FUNCTION_BLOCK FB_A_HKSystem IMPLEMENTS I_HKSystem
VAR_INPUT
	I_bVerbunden	:BOOL;		// Angabe ob HK-System angeschlossen ist
	I_iModus		:INT;		// Zustand des Systems (z.B. 0 = AUS | 1 = MAN | 2 = AUTO)
	I_iTemp			:INT;		// Aktuelle Temperatur um Heizmodus auszuwählen und zu stoppen
	I_bVerriegeln	:BOOL;		// Verriegelte Elemente sind nicht ansteuerbar
	I_bReset		:BOOL;		// Zustand des Baustein wird zurückgesetzt 
END_VAR

VAR_OUTPUT
	O_bPumpen		:BOOL;		// Pumpe des HK-Systems wird betrieben
	O_bKuehlen		:BOOL;		// HK-System heizt das Medium auf
	O_bHeizen		:BOOL;		// HK-System kühlt das Medium ab
	O_bStoerung		:BOOL;		// Befindet sich das Element in einem Error
	O_iStoerungID	:INT;		// Anzeigen von Störung über eine INT-Variable
	
END_VAR
	
VAR
	V_DefTemp		:INT;		// Variable für internes handling der Eigenschaft 
	V_Zeit			:TIME;		// Variable für internes handling der Eigenschaft 
	V_Zustand		:INT;		// Variable für internes handling der Eigenschaft 
	
	V_Timer			:TON;		// Runtime des Bausteins ermitteln
END_VAR

// Setzen der internen Variablen
V_Zeit := P_Laufzeit;
V_Zustand := P_Zustand;

// Fehler durch Verbindungsabbruch
IF O_bPumpen OR O_bKuehlen OR O_bHeizen THEN
	IF NOT I_bVerbunden THEN
		O_bPumpen := FALSE;
		O_bKuehlen := FALSE;
		O_bHeizen := FALSE;
		
		O_bStoerung := TRUE;
		O_iStoerungID := 04;
	END_IF
END_IF

// Abbruch des Heiz-Kühlprozesses beim erreichen der Temp
IF O_bHeizen OR O_bKuehlen THEN 
	IF I_iTemp = V_DefTemp THEN
		O_bKuehlen := FALSE;
		O_bHeizen := FALSE;		
	END_IF
END_IF

// Reset des Bausteins
IF I_bReset THEN
	O_bStoerung := FALSE;
	O_iStoerungID := 0;
END_IF

METHOD M_A_HK_AN : BOOL
VAR_INPUT
END_VAR
// EBENE 1: Verriegelung
IF NOT I_bVerriegeln THEN	
	// EBENE 2: AUTO-Modus
		IF I_iModus = 2 THEN
			// EBENE 3: Ist Pumpe AN
				IF O_bPumpen THEN
				// EBENE 4: Heizen oder Kühlen
					IF V_DefTemp > I_iTemp THEN
						O_bKuehlen := FALSE;
						O_bHeizen := TRUE;
						
						M_A_HK_AN := O_bHeizen;
						
					ELSIF I_iTemp > V_DefTemp THEN 	
						O_bHeizen := FALSE;
						O_bKuehlen := TRUE;
						
						M_A_HK_AN := O_bKuehlen;
					END_IF
				ELSE // Error: System ist nicht eingeschalten
					O_bStoerung := 1;
					O_iStoerungID := 11; 
				END_IF
			END_IF
END_IF
END_METHOD

METHOD M_A_HK_AUS : BOOL
VAR_INPUT
END_VAR
// EBENE 1: Verriegelung
IF NOT I_bVerriegeln THEN
		O_bKuehlen := FALSE;
		O_bHeizen := FALSE;
END_IF

IF O_bKuehlen = FALSE THEN
	M_A_HK_AUS := TRUE;
END_IF
END_METHOD

METHOD M_A_PUMPE_AN : BOOL
VAR_INPUT
END_VAR
// EBENE 1: Verriegelung
IF NOT I_bVerriegeln THEN	
	// EBENE 2: AUTO-Modus
		IF I_iModus = 2 THEN
			// EBENE 3: System muss angeschlossen sein
			IF I_bVerbunden THEN
				O_bPumpen := TRUE;
			ELSE 	// Error: System ist nicht angeschlossen
				O_bStoerung := 1;
				O_iStoerungID := 03;
			END_IF
		END_IF
END_IF

M_A_PUMPE_AN := O_bPumpen;
END_METHOD

METHOD M_A_PUMPE_AUS : BOOL
VAR_INPUT
END_VAR
// EBENE 1: Verriegelung
IF NOT I_bVerriegeln THEN
	IF NOT O_bHeizen AND NOT O_bKuehlen THEN
		O_bPumpen := FALSE;
	ELSE
		O_bStoerung := TRUE;
		O_iStoerungID := 05;
	END_IF
END_IF

IF O_bPumpen = FALSE THEN
	M_A_PUMPE_AUS := TRUE;
END_IF
END_METHOD

METHOD M_M_HK_AN : BOOL
VAR_INPUT
END_VAR
// EBENE 1: Verriegelung
IF NOT I_bVerriegeln THEN	
	// EBENE 2: MAN-Modus
		IF I_iModus = 1 THEN
			// EBENE 3: Ist Pumpe AN
				IF O_bPumpen THEN
				// EBENE 4: Heizen oder Kühlen
					IF V_DefTemp > I_iTemp THEN
						O_bKuehlen := FALSE;
						O_bHeizen := TRUE;
						
						M_M_HK_AN := O_bHeizen;
						
					ELSIF I_iTemp > V_DefTemp THEN 	
						O_bHeizen := FALSE;
						O_bKuehlen := TRUE;
						
						M_M_HK_AN := O_bKuehlen;
					END_IF
				ELSE // Error: System ist nicht eingeschalten
				O_bStoerung := 1;
				O_iStoerungID := 11; 	
				END_IF
			END_IF
END_IF
END_METHOD

METHOD M_M_HK_AUS : BOOL
VAR_INPUT
END_VAR
// EBENE 1: Verriegelung
IF NOT I_bVerriegeln THEN
		O_bKuehlen := FALSE;
		O_bHeizen := FALSE;
END_IF

IF O_bKuehlen = FALSE THEN
	M_M_HK_AUS := TRUE;
END_IF
END_METHOD

METHOD M_M_PUMPE_AN : BOOL
VAR_INPUT
END_VAR
// EBENE 1: Verriegelung
IF NOT I_bVerriegeln THEN	
	// EBENE 2: MAN-Modus
		IF I_iModus = 1 THEN
			// EBENE 3: System muss angeschlossen sein
			IF I_bVerbunden THEN
				O_bPumpen := TRUE;
			ELSE 	// Error: System ist nicht angeschlossen
				O_bStoerung := 1;
				O_iStoerungID := 03;
			END_IF
		END_IF
END_IF

M_M_PUMPE_AN := O_bPumpen;
END_METHOD

METHOD M_M_PUMPE_AUS : BOOL
VAR_INPUT
END_VAR
// EBENE 1: Verriegelung
IF NOT I_bVerriegeln THEN
	IF NOT O_bHeizen AND NOT O_bKuehlen THEN
		O_bPumpen := FALSE;
	ELSE
		O_bStoerung := TRUE;
		O_iStoerungID := 05;
	END_IF
END_IF

IF O_bPumpen = FALSE THEN
	M_M_PUMPE_AUS := TRUE;
END_IF
END_METHOD

PROPERTY P_DefTemp : INT
SET
END_SET
END_PROPERTY

PROPERTY P_Laufzeit : TIME
GET
IF O_bKuehlen OR O_bHeizen THEN
	V_Timer(IN := TRUE, PT := T#100H);
ELSE
	V_Timer(IN := FALSE);
END_IF

P_Laufzeit := V_Timer.ET;
END_GET
END_PROPERTY

PROPERTY PUBLIC P_Zustand : INT
GET
END_GET
END_PROPERTY

END_FUNCTION_BLOCK

(* stored: Version 1.1.0.1, ProductVersion 3.1.4024.12
   POU FB_A_HKSystem: Id {9fa8220f-7562-4362-b973-7f9818c39521}, SpecialFunc None
   Method M_A_HK_AN: Id {805f7cbf-a553-4d3b-9434-906e69543a3f}
   Method M_A_HK_AUS: Id {553ba116-732f-49c2-828c-c4f64984a7f1}
   Method M_A_PUMPE_AN: Id {27c2b7c0-1593-472c-8f45-d88c0777b443}
   Method M_A_PUMPE_AUS: Id {cae08f7a-6da2-419a-ab47-006b561ed974}
   Method M_M_HK_AN: Id {9431c962-da2e-4e6c-85e5-1e6aa4bd1568}
   Method M_M_HK_AUS: Id {edd300d5-3c05-4015-826d-b28d4c741cb4}
   Method M_M_PUMPE_AN: Id {14f6a021-156d-461b-8026-90385bcf155f}
   Method M_M_PUMPE_AUS: Id {111d2f64-fb00-4b2e-9656-c68c9627ae1f}
   Property P_DefTemp: Id {4c1a8e38-f9e9-47c1-a6a6-c8c687a40fad}
   Set Set: Id {3f98f9e9-b363-4a29-bea1-61c9c87b9f25}
   Property P_Laufzeit: Id {7f8750e8-fa8e-4ea4-b141-f777f59121ca}
   Get Get: Id {df4e3d5d-a935-4467-acce-4cb8897d6878}
   Property P_Zustand: Id {41e75813-f874-43a5-bfc6-f44385e63ae2}
   Get Get: Id {49cb2351-eb2a-4219-9220-c46d74796b7d} *)
